// TIA Portal project "FactoryIO_Template_S7-1200_V15_V17" (V17)
// Vorlageprojekt für das Buch mit Zielsystem S7-1200

(* hardware
DEVICE "S7-1200-Station_1"  S7-1200 Station
   slot 0: "Baugruppenträger_0"  Rack  V1.0
   slot 1: "PLC_1"  CPU 1214C DC/DC/Rly  6ES7 214-1HG40-0XB0  V4.5
   slot 2: "DQ 16x24VDC_1"  SM 1222 DQ16 x 24VDC  6ES7 222-1BH32-0XB0  V2.0
*)

// ===== PLC "PLC_1"  CPU 1214C DC/DC/Rly =====

VAR_GLOBAL   // PLC tag table "Standard-Variablentabelle"
   "START BUT" AT %I0.0 : Bool;
   "STOP BUT" AT %I0.1 : Bool;
   "RESET BUT" AT %I0.2 : Bool;
   "PALET SENSÖRÜ" AT %I0.3 : Bool;
   "ALT SENSÖR" AT %I0.4 : Bool;
   "ÜSTSENSÖRÜ" AT %I0.5 : Bool;
   "YÜKLENDİ SENSÖRÜ" AT %I0.6 : Bool;
   "SOL GİRİŞ SENSÖRÜ" AT %I0.7 : Bool;
   "SOL ÇIKIŞ SENSÖRÜ" AT %I1.0 : Bool;
   "SAĞ GİRİŞ SENSÖRÜ" AT %I1.1 : Bool;
   "SAĞ ÇIKIŞ SENSÖRÜ" AT %I1.2 : Bool;
   "ANA KONVEYÖR" AT %Q0.0 : Bool;
   "TRANSFER KONVEYÖRÜ" AT %Q0.1 : Bool;
   "SOLA TRANSFER" AT %Q0.2 : Bool;
   "SOL KONVEYÖR" AT %Q0.3 : Bool;
   "SAĞA TRANSFER" AT %Q0.4 : Bool;
   "SAĞ KONVEYÖR" AT %Q0.5 : Bool;
   "COUNTER EKRANI" AT %QW8 : Int;
   "START MEM" AT %M10.0 : Bool;
   "ALTSENSÖR MEM" AT %M10.1 : Bool;
   "YÜKLENDİSENSÖRMEM" AT %M10.2 : Bool;
   "ÜSTSENSÖR MEM" AT %M10.3 : Bool;
END_VAR

// folder: System blocks/Program resources

DATA_BLOCK "TİMER 1"   // DB1
{ S7_Optimized_Access := 'TRUE' }
AUTHOR : Simatic
FAMILY : IEC
NAME : IEC_TMR
VERSION : 1.0
// stored: InstanceOfName IEC_TIMER
"IEC_TIMER"
BEGIN
END_DATA_BLOCK

DATA_BLOCK "TİMER 2"   // DB2
{ S7_Optimized_Access := 'TRUE' }
AUTHOR : Simatic
FAMILY : IEC
NAME : IEC_TMR
VERSION : 1.0
// stored: InstanceOfName IEC_TIMER
"IEC_TIMER"
BEGIN
END_DATA_BLOCK

DATA_BLOCK "COUNTER"   // DB3
{ S7_Optimized_Access := 'TRUE' }
AUTHOR : Simatic
FAMILY : IEC
NAME : CNTR
VERSION : 1.0
// stored: InstanceOfName IEC_COUNTER
"IEC_COUNTER"
BEGIN
END_DATA_BLOCK

// folder: (top level)

FUNCTION "MHJ-PLC-Lab-Function-S71200" : Void   // FC9000, SCL
{ S7_Optimized_Access := 'TRUE' }
VERSION : 0.1
   VAR_TEMP
      rdTimeReturn : Int;
      outputTime : DTL;
      SyncVal : Byte;
      forVal : Int;
      forVal_2 : Int;
      Value : Byte;
   END_VAR
   VAR CONSTANT
      CompVal : Byte := 16#34;
      Value_01 : Byte := 16#11;
      Value_01_DW : DWord := 16#A165_D992;
      Value_02_DW : DWord := 16#58BE_4401;
   END_VAR
BEGIN

   #Value:=PEEK(area := 16#82,
        dbNumber := 0,
        byteOffset := 511);
   #Value := #Value + 1;

   POKE(area := 16#82,
        dbNumber := 0,
        byteOffset := 511,
        value := #Value);

   POKE(area:=16#81,
        dbNumber:=0,
        byteOffset:=1016,
        value:=#Value_01_DW);
   POKE(area := 16#81,
        dbNumber := 0,
        byteOffset := 1020,
        value := #Value_02_DW);

   POKE(area := 16#81,
        dbNumber := 0,
        byteOffset := 511,
        value := B#16#00);

   FOR #forVal := 0 TO 120 DO
       FOR #forVal_2:=0 TO 10 DO
           #rdTimeReturn:=RD_SYS_T(#outputTime);
           #rdTimeReturn := WR_SYS_T(#outputTime);
           #rdTimeReturn := RD_SYS_T(#outputTime);
           #rdTimeReturn := WR_SYS_T(#outputTime);
       END_FOR;
       #SyncVal:= PEEK(area := 16#81,
                      dbNumber := 0,
                      byteOffset := 511);
       IF #SyncVal = #CompVal THEN
          GOTO M_1;
       END_IF;
   END_FOR;
   RETURN;

   M_1:
   POKE(area := 16#81,
        dbNumber := 0,
        byteOffset := 511,
        value := B#16#0);
END_FUNCTION

ORGANIZATION_BLOCK "Main"   // OB1, LAD, ProgramCycle
TITLE = "Main Program Sweep (Cycle)"
{ S7_Optimized_Access := 'TRUE' }
VERSION : 0.1
   VAR_INPUT
      Initial_Call : Bool;   // Initial call of this OB
      Remanence : Bool;   // =True, if remanent data are available
   END_VAR
BEGIN

REGION Network 1: Konnektierungsbaustein für PLC-Lab
   // Im Netzwerk 1 wird der Konnektierungsbaustein für PLC-Lab aufgerufen.
   // Dieser Aufruf darf nicht entfernt werden!
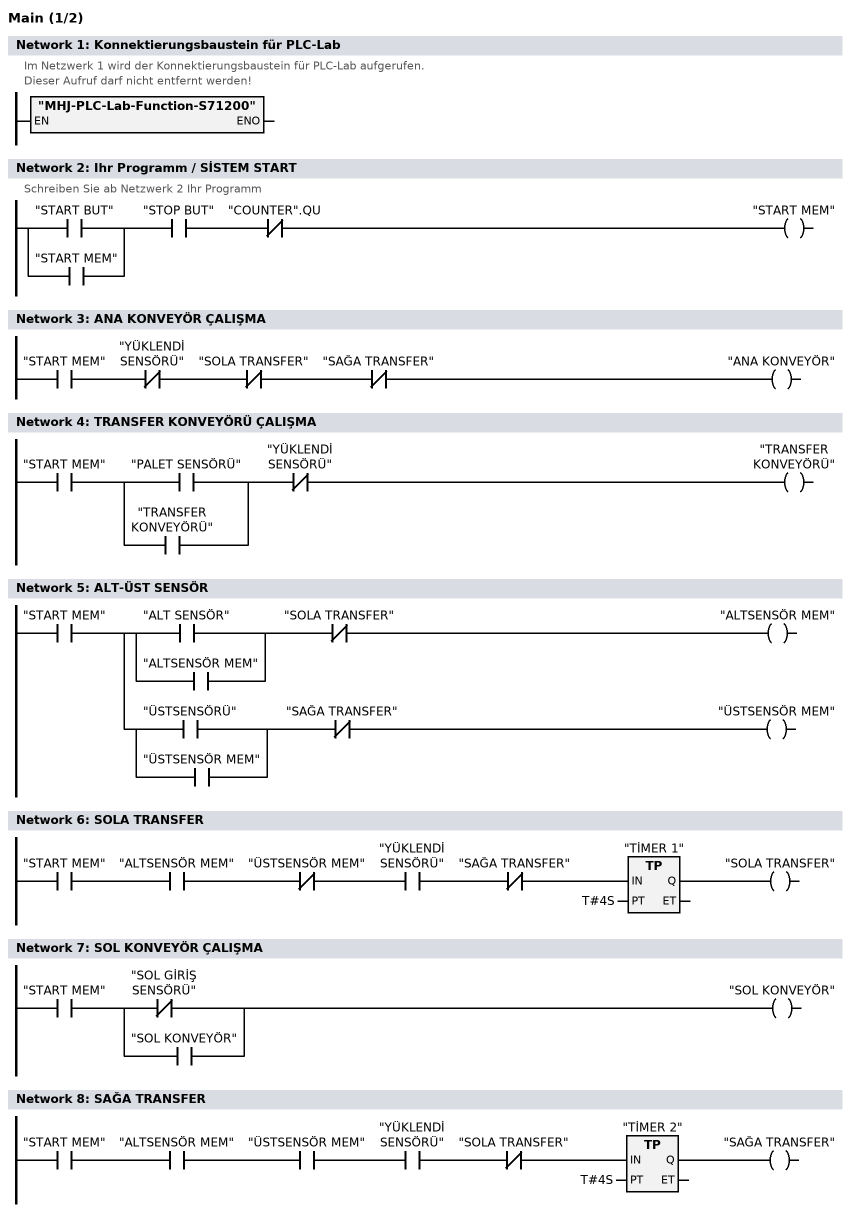
   RUNG wire#powerrail
      "MHJ-PLC-Lab-Function-S71200"()
   END_RUNG
   // the same network as SCL:
   "MHJ-PLC-Lab-Function-S71200"();
END_REGION

REGION Network 2: Ihr Programm / SİSTEM START
   // Schreiben Sie ab Netzwerk 2 Ihr Programm
   RUNG wire#powerrail
      Contact( "START BUT" )
      wire#w1
      Contact( "STOP BUT" )
      I_Contact( "COUNTER".QU )
      Coil( "START MEM" )
   END_RUNG
   RUNG wire#powerrail
      Contact( "START MEM" )
   END_RUNG wire#w1
   // the same network as SCL:
   "START MEM" := ("START BUT" OR "START MEM") AND "STOP BUT" AND NOT "COUNTER".QU;
END_REGION

REGION Network 3: ANA KONVEYÖR ÇALIŞMA
   RUNG wire#powerrail
      Contact( "START MEM" )
      I_Contact( "YÜKLENDİ SENSÖRÜ" )
      I_Contact( "SOLA TRANSFER" )
      I_Contact( "SAĞA TRANSFER" )
      Coil( "ANA KONVEYÖR" )
   END_RUNG
   // the same network as SCL:
   "ANA KONVEYÖR" := "START MEM" AND NOT "YÜKLENDİ SENSÖRÜ" AND NOT "SOLA TRANSFER" AND NOT "SAĞA TRANSFER";
END_REGION

REGION Network 4: TRANSFER KONVEYÖRÜ ÇALIŞMA
   RUNG wire#powerrail
      Contact( "START MEM" )
      wire#w1
      Contact( "PALET SENSÖRÜ" )
      wire#w2
      I_Contact( "YÜKLENDİ SENSÖRÜ" )
      Coil( "TRANSFER KONVEYÖRÜ" )
   END_RUNG
   RUNG wire#w1
      Contact( "TRANSFER KONVEYÖRÜ" )
   END_RUNG wire#w2
   // the same network as SCL:
   "TRANSFER KONVEYÖRÜ" := "START MEM" AND ("PALET SENSÖRÜ" OR "TRANSFER KONVEYÖRÜ") AND NOT "YÜKLENDİ SENSÖRÜ";
END_REGION

REGION Network 5: ALT-ÜST SENSÖR
   RUNG wire#powerrail
      Contact( "START MEM" )
      wire#w1
      Contact( "ALT SENSÖR" )
      wire#w2
      I_Contact( "SOLA TRANSFER" )
      Coil( "ALTSENSÖR MEM" )
   END_RUNG
   RUNG wire#w1
      Contact( "ALTSENSÖR MEM" )
   END_RUNG wire#w2
   RUNG wire#w1
      Contact( "ÜSTSENSÖRÜ" )
      wire#w3
      I_Contact( "SAĞA TRANSFER" )
      Coil( "ÜSTSENSÖR MEM" )
   END_RUNG
   RUNG wire#w1
      Contact( "ÜSTSENSÖR MEM" )
   END_RUNG wire#w3
   // the same network as SCL:
   "ALTSENSÖR MEM" := "START MEM" AND ("ALT SENSÖR" OR "ALTSENSÖR MEM") AND NOT "SOLA TRANSFER";
   "ÜSTSENSÖR MEM" := "START MEM" AND ("ÜSTSENSÖRÜ" OR "ÜSTSENSÖR MEM") AND NOT "SAĞA TRANSFER";
END_REGION

REGION Network 6: SOLA TRANSFER
   "TİMER 1".TP(IN := "START MEM" AND "ALTSENSÖR MEM" AND NOT "ÜSTSENSÖR MEM" AND "YÜKLENDİ SENSÖRÜ" AND NOT "SAĞA TRANSFER",
                PT := T#4S);
   "SOLA TRANSFER" := "TİMER 1".Q;
END_REGION

REGION Network 7: SOL KONVEYÖR ÇALIŞMA
   RUNG wire#powerrail
      Contact( "START MEM" )
      wire#w1
      I_Contact( "SOL GİRİŞ SENSÖRÜ" )
      wire#w2
      Coil( "SOL KONVEYÖR" )
   END_RUNG
   RUNG wire#w1
      Contact( "SOL KONVEYÖR" )
   END_RUNG wire#w2
   // the same network as SCL:
   "SOL KONVEYÖR" := "START MEM" AND (NOT "SOL GİRİŞ SENSÖRÜ" OR "SOL KONVEYÖR");
END_REGION

REGION Network 8: SAĞA TRANSFER
   "TİMER 2".TP(IN := "START MEM" AND "ALTSENSÖR MEM" AND "ÜSTSENSÖR MEM" AND "YÜKLENDİ SENSÖRÜ" AND NOT "SOLA TRANSFER",
                PT := T#4S);
   "SAĞA TRANSFER" := "TİMER 2".Q;
END_REGION

REGION Network 9: SAĞ KONVEYÖR
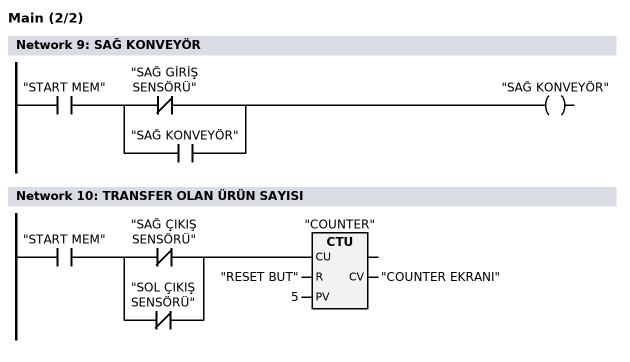
   RUNG wire#powerrail
      Contact( "START MEM" )
      wire#w1
      I_Contact( "SAĞ GİRİŞ SENSÖRÜ" )
      wire#w2
      Coil( "SAĞ KONVEYÖR" )
   END_RUNG
   RUNG wire#w1
      Contact( "SAĞ KONVEYÖR" )
   END_RUNG wire#w2
   // the same network as SCL:
   "SAĞ KONVEYÖR" := "START MEM" AND (NOT "SAĞ GİRİŞ SENSÖRÜ" OR "SAĞ KONVEYÖR");
END_REGION

REGION Network 10: TRANSFER OLAN ÜRÜN SAYISI
   "COUNTER".CTU(CU := "START MEM" AND (NOT "SAĞ ÇIKIŞ SENSÖRÜ" OR NOT "SOL ÇIKIŞ SENSÖRÜ"),
                 R := "RESET BUT",
                 PV := 5,
                 CV => "COUNTER EKRANI");
END_REGION
END_ORGANIZATION_BLOCK